FUNCTION_BLOCK FB_RollingAverageConsumer
VAR
    adder : B1RollingAverage_Plc.FB_RollingAverage;
    lastResult : INT;
END_VAR

lastResult := adder.Step(sample := 10);

END_FUNCTION_BLOCK

(* stored: Version 1.1.0.1
   POU FB_RollingAverageConsumer: Id {d09f4244-e47f-4e29-b442-c50bc18fe19d}, SpecialFunc None *)
